Yaskawa INFORM job: FRONT_WELD_-90ST-2_5140.JBI

/JOB
//NAME FRONT_WELD_-90ST-2_5140
///FOLDERNAME 02-SKRZYNIE_JOBS
//POS
///NPOS 31,31,0,6,0,0
///TOOL 0
///POSTYPE PULSE
///PULSE
C00000=0,-52278,40443,0,6873,-1
C00001=0,-52278,40443,0,6873,-1
C00002=0,-42686,23640,-7425,-34877,-70985
C00003=-25126,-44577,-4813,-57071,-34461,-49771
C00004=-6017,-48449,-29001,-102269,-8383,-26407
C00005=-2863,-32693,-8619,-87056,-6043,-33280
C00006=-4454,-30190,-5337,-84437,-7079,-34689
C00007=-4440,-30147,-5223,-84074,-7073,-34859
C00008=6049,-30496,-6078,-83018,-361,-34269
C00009=23053,-29108,-5505,-81506,10657,-33192
C00010=32667,-27182,-4171,-80231,16911,-32822
C00011=43283,-23925,-1748,-78590,23862,-32556
C00012=50847,-28145,-10545,-73666,29314,-34422
C00013=73589,-4766,14825,-76336,20345,-43289
C00014=77780,4684,28307,-81126,26309,-43327
C00015=77759,4649,28267,-81123,26295,-43330
C00016=74815,1594,24890,-81179,24551,-43729
C00017=78305,2073,15702,-60453,36425,-62227
C00018=70502,-5550,9869,-62064,28728,-60210
C00019=59595,-12633,6156,-66364,18535,-56886
C00020=58678,-17366,4552,-88847,13968,-42180
C00021=-23545,-30165,-21390,-32579,21562,-60781
C00022=-43411,-19640,-10965,1347,18370,-78573
C00023=-46554,-16064,-6940,7268,18455,-81640
C00024=-53996,-17904,-12508,38045,33194,-82968
C00025=-40513,-24909,-18256,27984,27249,-76648
C00026=-27124,-28543,-20634,12993,23111,-67991
C00027=-24971,-35737,-30976,9397,24510,-66000
C00028=0,-42686,23640,-7425,-34877,-70985
C00029=0,-52278,40443,-5610,-49281,-72137
C00030=0,-52278,40443,0,6873,-1
BC00000=760319
BC00001=790120
BC00002=918401
BC00003=956036
BC00004=986861
BC00005=986861
BC00006=986864
BC00007=986864
BC00008=986863
BC00009=986862
BC00010=986862
BC00011=986862
BC00012=986862
BC00013=986863
BC00014=986863
BC00015=986863
BC00016=986861
BC00017=986863
BC00018=986863
BC00019=986863
BC00020=986863
BC00021=986863
BC00022=986862
BC00023=986862
BC00024=986860
BC00025=986861
BC00026=986862
BC00027=986862
BC00028=918401
BC00029=790120
BC00030=790120
///POSTYPE BASE
///RECTAN
///RCONF 1,0,0,0,0,0,0,0,0,0,0,0,0,0,0,0,0,0,0,0,0,0,0,0
P00500=2.332,-5.281,-1.258,0.0000,0.0000,0.0000
///RCONF 0,0,0,0,0,0,0,0,0,0,0,0,0,0,0,0,0,0,0,0,0,0,0,0
P00501=-2.026,0.009,3.534,0.0000,0.0000,0.0000
///RCONF 1,0,0,0,0,0,0,0,0,0,0,0,0,0,0,0,0,0,0,0,0,0,0,0
P00502=-2.023,0.001,1.732,0.0000,0.0000,0.0000
P00503=0.138,-0.044,1.539,0.0000,0.0000,0.0000
P00504=-0.309,-0.010,1.636,0.0000,0.0000,0.0000
P00505=0.999,-9.916,8.214,0.0000,0.0000,0.0000
//INST
///DATE 2024/06/04 21:12
///ATTR SC,RW
///GROUP1 RB1,BS1
NOP
MOVJ C00000 BC00000 VJ=60.00
MOVJ C00001 BC00001 VJ=60.00
MOVJ C00002 BC00002 VJ=60.00
MOVJ C00003 BC00003 VJ=60.00
MOVJ C00004 BC00004 VJ=30.00
'::::::::::::::::::::::::::::::::
'W20
'::::::::::::::::::::::::::::::::
MOVL C00005 BC00005 V=500.0
SFTON P0503
MACRO1 MJ#(0) ARGF14
MOVL C00006 BC00006 V=166.7 PL=0
ARCON
MOVC C00007 BC00007 V=9.5
MOVC C00008 BC00008 V=9.5
MOVC C00009 BC00009 V=9.5
SFTOF
SFTON P0502
MOVC C00010 BC00010 V=9.5
MOVC C00011 BC00011 V=9.5
ARCOF
MOVL C00012 BC00012 V=166.7
SFTOF
'::::::::::::::::::::::::::::::::
'W21
'::::::::::::::::::::::::::::::::
MOVL C00013 BC00013 V=333.3
SFTON P0500
MACRO1 MJ#(0) ARGF14
MOVL C00014 BC00014 V=166.7 PL=0
ARCON
MOVC C00015 BC00015 V=9.5
MOVC C00016 BC00016 V=9.5
MOVC C00017 BC00017 V=9.5
SFTOF
SFTON P0501
MOVC C00018 BC00018 V=9.5
MOVC C00019 BC00019 V=9.5
ARCOF
MOVL C00020 BC00020 V=166.7
SFTOF
MOVL C00021 BC00021 V=500.0
'::::::::::::::::::::::::::::::::
'W22
'::::::::::::::::::::::::::::::::
MOVL C00022 BC00022 V=500.0
SFTON P0505
MACRO1 MJ#(0) ARGF14
MOVL C00023 BC00023 V=166.7 PL=0
ARCON
MOVL C00024 BC00024 V=10.0
SFTOF
SFTON P0504
MOVL C00025 BC00025 V=9.5
MOVL C00026 BC00026 V=10.0
ARCOF
MOVL C00027 BC00027 V=333.3
SFTOF
MOVJ C00028 BC00028 VJ=70.00
MOVJ C00029 BC00029 VJ=80.00
MOVJ C00030 BC00030 VJ=80.00
END
